
FUNCTION CB_lt_time : BOOL


TITLE = ' Test Whether IN0 is strictly less than IN1 '
VERSION : '1.0'
AUTHOR  : CB
NAME    : lt_time
FAMILY  : TNI

VAR_INPUT
    IN0 : TIME;
    IN1 : TIME;
END_VAR

BEGIN

CB_lt_time := (IN0 < IN1);

END_FUNCTION
